// Element Shuttle car with forks inputs
TYPE ST_HW_Inputs_Conv_ShuttleForks EXTENDS ST_HW_InputsMPD_Conv :

STRUCT	
END_STRUCT
END_TYPE

(* stored: Version 1.1.0.1, ProductVersion 3.1.4024.9
   DUT ST_HW_Inputs_Conv_ShuttleForks: Id {0f56ecc4-7768-47d6-9731-9522111d51b3} *)
